(* CoDeSys 2.3.9.35 project: PACMAN.pro *)
(* Libraries: Util_no_Real.lib 1.6.07 09:41:00, Standard.LIB 4.10.05 11:14:46 *)

(* Global variable list: Global_Variables *)
VAR_GLOBAL
    hoz: INT;
    ver: INT;
	MAPA: ARRAY[0..20, 0..15] OF BOOL;
	Mapa_Punkty: ARRAY[0..20, 0..15] OF BOOL;
	Wolne_Prawo: BOOL;
	Wolne_Lewo: BOOL;
	Wolne_Dol: BOOL;
	Wolne_Gora: BOOL;
	Otwarte: BOOL := TRUE;
	Kierunek: INT := 1;
 B_Prawo : BOOL := TRUE;
   B_Lewo  : BOOL;
   B_Dol   : BOOL;
   B_Gora  : BOOL;

END_VAR

(* POU PLC_PRG, LD *)
PROGRAM PLC_PRG
VAR
	S1: BOOL;
	S3: BOOL;
	res: BOOL;
	S2: BOOL;
	S4: BOOL;
	C3: CTUD;
	W1: BOOL;
	C4: CTUD;
	Ruch_Lewo: BOOL;
	Ruch_Dol: BOOL;
	DUMMY: BOOL;
	M1:MAPA;
	Ruch_Gora: BOOL;
	T_Ani: TON;
	C_Ani: CTU;
	SR1: SR;
	Reset_SR1: BOOL;
	SR2: SR;
	Reset_SR2: BOOL;
	SR3: SR;
	Reset_SR3: BOOL;
	Reset_SR4: BOOL;
	SR4: SR;
	T_Ruch: TON;
END_VAR
_LD_ (* Ladder Diagram *)
NETWORK 1
	M1:MAPA()
NETWORK 2
	*
		EN --- ???:OBLICZ_KOLIZJE() => DUMMY
NETWORK 3
	[/T_Ruch.Q] - T_Ruch:TON(IN: *, PT: T#200ms)
NETWORK 4
	[/T_Ruch.Q] - [B_Dol] - [Wolne_Dol] - C3:CTUD(CU: *, CD: Ruch_Gora, RESET: res, LOAD: FALSE, PV: 20, CV => ver)
NETWORK 5
	[/T_Ruch.Q] - [B_Gora] - [Wolne_Gora] --- (Ruch_Gora)
NETWORK 6
	[/T_Ruch.Q] - [B_Prawo] - [Wolne_Prawo] - C4:CTUD(CU: *, CD: Ruch_Lewo, RESET: res, LOAD: FALSE, PV: 15, CV => hoz)
NETWORK 7
	[/T_Ruch.Q] - [B_Lewo] - [Wolne_Lewo] --- (Ruch_Lewo)
NETWORK 8
	[/T_Ani.Q] - T_Ani:TON(IN: *, PT: T#20ms)
NETWORK 9
	[T_Ani.Q] - C_Ani:CTU(CU: *, RESET: C_Ani.Q, PV: 2)
NETWORK 10
	[/C_Ani.CV.0] --- (Otwarte)
NETWORK 11
	[S1] - SR1:SR(SET1: *, RESET: Reset_SR1) --- (B_Prawo)
NETWORK 12
	{ [S2] | [S3] | [S4] } --- (Reset_SR1)
NETWORK 13
	[S2] - SR2:SR(SET1: *, RESET: Reset_SR2) --- (B_Lewo)
NETWORK 14
	{ [S1] | [S3] | [S4] } --- (Reset_SR2)
NETWORK 15
	[S3] - SR3:SR(SET1: *, RESET: Reset_SR3) --- (B_Dol)
NETWORK 16
	{ [S1] | [S2] | [S4] } --- (Reset_SR3)
NETWORK 17
	[S4] - SR4:SR(SET1: *, RESET: Reset_SR4) --- (B_Gora)
NETWORK 18
	{ [S1] | [S2] | [S3] } --- (Reset_SR4)
NETWORK 19
	[Mapa_Punkty[hoz, ver]] --- (R Mapa_Punkty[hoz, ver])
_END_LD_
(* the same logic as Structured Text *)
(* Network 1 *)
M1();
(* Network 2: see the listing above *)
(* Network 3 *)
T_Ruch(IN := NOT T_Ruch.Q, PT := T#200ms);
(* Network 4 *)
C3(CU := NOT T_Ruch.Q AND B_Dol AND Wolne_Dol, CD := Ruch_Gora, RESET := res, LOAD := FALSE, PV := 20);
ver := C3.CV;
(* Network 5 *)
Ruch_Gora := NOT T_Ruch.Q AND B_Gora AND Wolne_Gora;
(* Network 6 *)
C4(CU := NOT T_Ruch.Q AND B_Prawo AND Wolne_Prawo, CD := Ruch_Lewo, RESET := res, LOAD := FALSE, PV := 15);
hoz := C4.CV;
(* Network 7 *)
Ruch_Lewo := NOT T_Ruch.Q AND B_Lewo AND Wolne_Lewo;
(* Network 8 *)
T_Ani(IN := NOT T_Ani.Q, PT := T#20ms);
(* Network 9 *)
C_Ani(CU := T_Ani.Q, RESET := C_Ani.Q, PV := 2);
(* Network 10 *)
Otwarte := NOT C_Ani.CV.0;
(* Network 11 *)
SR1(SET1 := S1, RESET := Reset_SR1);
B_Prawo := SR1.Q1;
(* Network 12 *)
Reset_SR1 := S2 OR S3 OR S4;
(* Network 13 *)
SR2(SET1 := S2, RESET := Reset_SR2);
B_Lewo := SR2.Q1;
(* Network 14 *)
Reset_SR2 := S1 OR S3 OR S4;
(* Network 15 *)
SR3(SET1 := S3, RESET := Reset_SR3);
B_Dol := SR3.Q1;
(* Network 16 *)
Reset_SR3 := S1 OR S2 OR S4;
(* Network 17 *)
SR4(SET1 := S4, RESET := Reset_SR4);
B_Gora := SR4.Q1;
(* Network 18 *)
Reset_SR4 := S1 OR S2 OR S3;
(* Network 19 *)
IF Mapa_Punkty[hoz, ver] THEN Mapa_Punkty[hoz, ver] := FALSE; END_IF;
END_PROGRAM

(* POU MAPA, ST *)
FUNCTION_BLOCK MAPA
VAR
    i: INT;
    j: INT;
    Init_Done: BOOL := FALSE;

END_VAR
IF NOT Init_Done THEN

    (* ======================= *)
    (* 1. RYSOWANIE ŒCIAN      *)
    (* ======================= *)

    FOR i := 0 TO 20 DO
        Mapa[i, 0] := TRUE;
        Mapa[i, 15] := TRUE;
    END_FOR
    
    FOR j := 0 TO 15 DO
        Mapa[0, j] := TRUE;
        MAPA[20, j] := TRUE;
    END_FOR

    Mapa[0, 0] := FALSE;
    Mapa[1, 0] := FALSE;
    Mapa[0, 1] := FALSE;
    Mapa[2, 0] := FALSE;
    Mapa[0, 2] := FALSE;
    Mapa[3, 0] := FALSE;
    Mapa[0, 3] := FALSE;
    Mapa[0, 4] := FALSE;
    Mapa[0, 5] := FALSE;
    Mapa[0, 6] := FALSE;
    Mapa[0, 7] := FALSE;
    Mapa[0, 8] := FALSE;

    Mapa[1, 4] := FALSE;
    Mapa[2, 4] := FALSE;
    Mapa[2, 3] := FALSE;
    Mapa[2, 2] := FALSE;
    Mapa[3, 2] := FALSE;
    
    Mapa[1, 3] := TRUE;
    Mapa[1, 2] := TRUE;
    Mapa[1, 1] := TRUE;
    Mapa[2, 1] := TRUE;

    Mapa[1, 5] := TRUE;
    Mapa[1, 6] := TRUE;
    Mapa[1, 7] := TRUE;
    Mapa[2, 7] := TRUE;
    Mapa[3, 5] := TRUE;
    Mapa[4, 5] := TRUE;
    Mapa[3, 3] := TRUE;
    Mapa[4, 3] := TRUE;
    Mapa[4, 7] := TRUE;
    Mapa[4, 8] := TRUE;

    Mapa[6, 1] := TRUE;
    Mapa[7, 1] := TRUE;
    Mapa[8, 1] := TRUE;
    Mapa[9, 1] := TRUE;
    Mapa[10, 1] := TRUE;
    Mapa[11, 1] := TRUE;
    Mapa[12, 1] := TRUE;

    Mapa[6, 3] := TRUE;
    Mapa[7, 3] := TRUE;
    Mapa[11, 3] := TRUE;
    Mapa[12, 3] := TRUE;
    Mapa[6, 4] := TRUE;
    Mapa[12, 4] := TRUE;

    Mapa[6, 5] := TRUE;
    Mapa[7, 5] := TRUE;
    Mapa[8, 5] := TRUE;
    Mapa[9, 5] := TRUE;
    Mapa[10, 5] := TRUE;
    Mapa[11, 5] := TRUE;
    Mapa[12, 5] := TRUE;

    Mapa[6, 7] := TRUE;
    Mapa[7, 7] := TRUE;
    Mapa[8, 7] := TRUE;
    Mapa[9, 7] := TRUE;
    Mapa[10, 7] := TRUE;
    Mapa[11, 7] := TRUE;
    Mapa[12, 7] := TRUE;

    Mapa[14, 0] := TRUE;
    Mapa[14, 1] := TRUE;
    Mapa[14, 3] := TRUE;
    Mapa[14, 5] := TRUE;
    Mapa[15, 5] := TRUE;
    Mapa[14, 7] := TRUE;
    Mapa[14, 8] := TRUE;
    Mapa[15, 3] := TRUE;
    Mapa[16, 1] := TRUE;
    Mapa[16, 7] := TRUE;

    Mapa[17, 1] := TRUE;
    Mapa[17, 2] := TRUE;
    Mapa[17, 3] := TRUE;
    Mapa[17, 5] := TRUE;
    Mapa[17, 6] := TRUE;
    Mapa[17, 7] := TRUE;
    
    Mapa[4, 1] := TRUE;

    Mapa[5, 0] := FALSE;
    Mapa[6, 0] := FALSE;
    Mapa[7, 0] := FALSE;
    Mapa[8, 0] := FALSE;
    Mapa[9, 0] := FALSE;
    Mapa[10, 0] := FALSE;
    Mapa[11, 0] := FALSE;
    Mapa[12, 0] := FALSE;
    Mapa[13, 0] := FALSE;
    Mapa[15, 0] := FALSE;
    Mapa[16, 0] := FALSE;
    Mapa[17, 0] := FALSE;
    Mapa[18, 0] := FALSE;


    Mapa[1, 9] := TRUE;
    Mapa[2, 9] := TRUE;
    Mapa[3, 9] := TRUE;
    Mapa[4, 9] := TRUE;
    Mapa[5, 9] := TRUE;
    Mapa[6, 9] := TRUE;
    Mapa[7, 9] := TRUE;
    Mapa[8, 9] := TRUE;
    Mapa[9, 9] := TRUE;
    Mapa[10, 9] := TRUE;
    Mapa[11, 9] := TRUE;
    Mapa[12, 9] := TRUE;
    Mapa[13, 9] := TRUE;
    Mapa[14, 9] := TRUE;
    Mapa[15, 9] := TRUE;
    Mapa[16, 9] := TRUE;
    Mapa[17, 9] := TRUE;
    Mapa[18, 9] := TRUE;
    Mapa[19, 9] := TRUE;

    Mapa[19, 1] := TRUE;
    Mapa[19, 2] := TRUE;
    Mapa[19, 3] := TRUE;
    Mapa[19, 4] := TRUE;
    Mapa[19, 5] := TRUE;
    Mapa[19, 6] := TRUE;
    Mapa[19, 7] := TRUE;
    Mapa[19, 8] := TRUE;

    (* ======================= *)
    (* 2. RYSOWANIE PUNKTÓW    *)
    (* ======================= *)
    
	Mapa_Punkty[0, 2] := TRUE;
	Mapa_Punkty[0, 3] := TRUE;
	Mapa_Punkty[0, 4] := TRUE;
	Mapa_Punkty[0, 5] := TRUE;
	Mapa_Punkty[0, 6] := TRUE;
	Mapa_Punkty[0, 7] := TRUE;
	Mapa_Punkty[0, 8] := TRUE;
	Mapa_Punkty[1, 8] := TRUE;
	Mapa_Punkty[2, 8] := TRUE;
	Mapa_Punkty[3, 8] := TRUE;
	Mapa_Punkty[3, 7] := TRUE;
	Mapa_Punkty[3, 6] := TRUE;
	Mapa_Punkty[4, 6] := TRUE;
	Mapa_Punkty[5, 6] := TRUE;
	Mapa_Punkty[6, 6] := TRUE;
	Mapa_Punkty[7, 6] := TRUE;
	Mapa_Punkty[8, 6] := TRUE;
	Mapa_Punkty[9, 6] := TRUE;
	Mapa_Punkty[10, 6] := TRUE;
	Mapa_Punkty[11,6] := TRUE;
	Mapa_Punkty[12, 6] := TRUE;
	Mapa_Punkty[13, 6] := TRUE;
	Mapa_Punkty[14, 6] := TRUE;
	Mapa_Punkty[15, 6] := TRUE;
	Mapa_Punkty[16, 6] := TRUE;
	
	Mapa_Punkty[6, 8] := TRUE;
	Mapa_Punkty[7, 8] := TRUE;
	Mapa_Punkty[8, 8] := TRUE;
	Mapa_Punkty[9, 8] := TRUE;
	Mapa_Punkty[10, 8] := TRUE;
	Mapa_Punkty[11, 8] := TRUE;
	Mapa_Punkty[12, 8] := TRUE;
	Mapa_Punkty[13, 8] := TRUE;
	Mapa_Punkty[5, 8] := TRUE;
	
	Mapa_Punkty[6, 0] := TRUE;
	Mapa_Punkty[7, 0] := TRUE;
	Mapa_Punkty[8, 0] := TRUE;
	Mapa_Punkty[9, 0] := TRUE;
	Mapa_Punkty[10, 0] := TRUE;
	Mapa_Punkty[11, 0] := TRUE;
	Mapa_Punkty[12, 0] := TRUE;
	Mapa_Punkty[13, 0] := TRUE;
	Mapa_Punkty[5, 0] := TRUE;
	
	Mapa_Punkty[18, 0] := TRUE;
	Mapa_Punkty[18, 1] := TRUE;
	Mapa_Punkty[18, 2] := TRUE;
	Mapa_Punkty[18, 3] := TRUE;
	Mapa_Punkty[18, 4] := TRUE;
	Mapa_Punkty[18, 5] := TRUE;
	Mapa_Punkty[18, 6] := TRUE;
	Mapa_Punkty[18, 7] := TRUE;
	Mapa_Punkty[18, 8] := TRUE;
	
	Mapa_Punkty[2, 2] := TRUE;
	Mapa_Punkty[3, 2] := TRUE;
	Mapa_Punkty[4, 2] := TRUE;
	Mapa_Punkty[5, 2] := TRUE;
	Mapa_Punkty[6, 2] := TRUE;
	Mapa_Punkty[7, 2] := TRUE;
	Mapa_Punkty[8, 2] := TRUE;
	Mapa_Punkty[9, 2] := TRUE;
	Mapa_Punkty[10, 2] := TRUE;
	Mapa_Punkty[11, 2] := TRUE;
	Mapa_Punkty[12, 2] := TRUE;
	Mapa_Punkty[13, 2] := TRUE;
	Mapa_Punkty[14, 2] := TRUE;
	Mapa_Punkty[15, 2] := TRUE;
	Mapa_Punkty[16, 2] := TRUE;
	
	Mapa_Punkty[2, 3] := TRUE;
	Mapa_Punkty[2, 4] := TRUE;
	Mapa_Punkty[2, 5] := TRUE;
	Mapa_Punkty[2, 6] := TRUE;
	
	Mapa_Punkty[5, 0] := TRUE;
	Mapa_Punkty[5, 1] := TRUE;
	Mapa_Punkty[5, 3] := TRUE;
	Mapa_Punkty[5, 4] := TRUE;
	Mapa_Punkty[5, 5] := TRUE;
	Mapa_Punkty[5, 7] := TRUE;
	Mapa_Punkty[5, 8] := TRUE;
	Mapa_Punkty[3, 4] := TRUE;
	Mapa_Punkty[4, 4] := TRUE;
	
	Mapa_Punkty[8, 3] := TRUE;
	Mapa_Punkty[9, 3] := TRUE;
	Mapa_Punkty[10, 3] := TRUE;
	
	Mapa_Punkty[7,4] := TRUE;
	Mapa_Punkty[8,4] := TRUE;
	Mapa_Punkty[9,4] := TRUE;
	Mapa_Punkty[10,4] := TRUE;
	Mapa_Punkty[11,4] := TRUE;
	
	Mapa_Punkty[13,1] := TRUE;
	Mapa_Punkty[13,3] := TRUE;
	Mapa_Punkty[13,4] := TRUE;
	Mapa_Punkty[13,5] := TRUE;
	Mapa_Punkty[13,7] := TRUE;
	
	Mapa_Punkty[13,4] := TRUE;
	Mapa_Punkty[14,4] := TRUE;
	Mapa_Punkty[15,4] := TRUE;
	Mapa_Punkty[16,4] := TRUE;
	Mapa_Punkty[17,4] := TRUE;
	
	Mapa_Punkty[16,3] := TRUE;
	Mapa_Punkty[16,5] := TRUE;
	
	Mapa_Punkty[15,0] := TRUE;
	Mapa_Punkty[16,0] := TRUE;
	Mapa_Punkty[17,0] := TRUE;
	Mapa_Punkty[15,8] := TRUE;
	Mapa_Punkty[16,8] := TRUE;
	Mapa_Punkty[17,8] := TRUE;
	Mapa_Punkty[15,1] := TRUE;
	Mapa_Punkty[1,4] := TRUE;
	Mapa_Punkty[15,7] := TRUE;
	
	Mapa_Punkty[1,0] := TRUE;
	Mapa_Punkty[2,0] := TRUE;
	Mapa_Punkty[3,0] := TRUE;
	Mapa_Punkty[3,1] := TRUE;

    Init_Done := TRUE;

END_IF
END_FUNCTION_BLOCK

(* POU OBLICZ_KOLIZJE, ST *)
PROGRAM OBLICZ_KOLIZJE
VAR
END_VAR
Wolne_Prawo := FALSE;
Wolne_Lewo := FALSE;
Wolne_Gora := FALSE;
Wolne_Dol := FALSE;

IF hoz < 20 THEN
    IF Mapa[hoz + 1, ver] = FALSE THEN
        Wolne_Prawo := TRUE;
    END_IF
END_IF


IF hoz > 0 THEN
    IF Mapa[hoz - 1, ver] = FALSE THEN
        Wolne_Lewo := TRUE;
    END_IF
END_IF

IF ver < 15 THEN
    IF Mapa[hoz, ver + 1] = FALSE THEN
        Wolne_Dol := TRUE;
    END_IF
END_IF

IF ver > 0 THEN
    IF Mapa[hoz, ver - 1] = FALSE THEN
        Wolne_Gora := TRUE;
    END_IF
END_IF
END_PROGRAM

(* Visualisation GRA
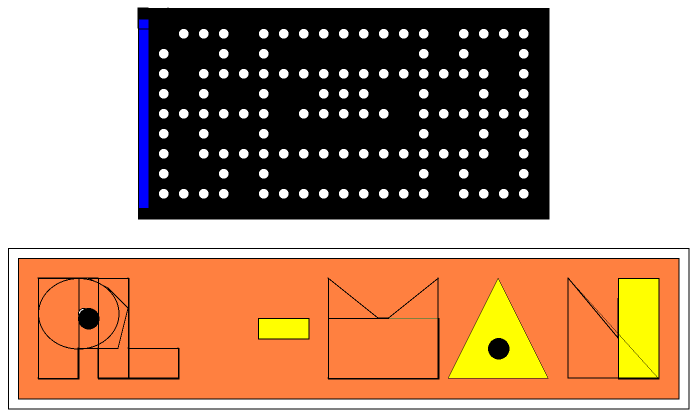
ellipse at (180,150)-(191,161): invisible if NOT Mapa_Punkty[0, 1]
ellipse at (180,190)-(191,201): invisible if NOT Mapa_Punkty[0, 3]
ellipse at (180,210)-(191,221): invisible if NOT Mapa_Punkty[0, 4]
ellipse at (180,230)-(191,241): invisible if NOT Mapa_Punkty[0,5]
ellipse at (180,250)-(191,261): invisible if NOT Mapa_Punkty[0,6]
ellipse at (180,270)-(191,281): invisible if NOT Mapa_Punkty[0,7]
ellipse at (180,290)-(191,301): invisible if NOT Mapa_Punkty[0,8]
ellipse at (200,290)-(211,301): invisible if NOT Mapa_Punkty[1,8]
ellipse at (220,290)-(231,301): invisible if NOT Mapa_Punkty[2,8]
ellipse at (240,290)-(251,301): invisible if NOT Mapa_Punkty[3,8]
ellipse at (240,270)-(251,281): invisible if NOT Mapa_Punkty[3,7]
ellipse at (240,250)-(251,261): invisible if NOT Mapa_Punkty[3,6]
ellipse at (220,250)-(231,261): invisible if NOT Mapa_Punkty[2,6]
ellipse at (260,250)-(271,261): invisible if NOT Mapa_Punkty[4,6]
ellipse at (280,250)-(291,261): invisible if NOT Mapa_Punkty[5,6]
ellipse at (300,250)-(311,261): invisible if NOT Mapa_Punkty[6,6]
ellipse at (320,250)-(331,261): invisible if NOT Mapa_Punkty[7,6]
ellipse at (340,250)-(351,261): invisible if NOT Mapa_Punkty[8,6]
ellipse at (360,250)-(371,261): invisible if NOT Mapa_Punkty[9,6]
ellipse at (380,250)-(391,261): invisible if NOT Mapa_Punkty[10,6]
ellipse at (400,250)-(411,261): invisible if NOT Mapa_Punkty[11,6]
ellipse at (420,250)-(431,261): invisible if NOT Mapa_Punkty[12,6]
ellipse at (440,250)-(451,261): invisible if NOT Mapa_Punkty[13,6]
ellipse at (460,250)-(471,261): invisible if NOT Mapa_Punkty[14,6]
ellipse at (480,250)-(491,261): invisible if NOT Mapa_Punkty[15,6]
ellipse at (500,250)-(511,261): invisible if NOT Mapa_Punkty[16,6]
ellipse at (280,290)-(291,301): invisible if NOT Mapa_Punkty[5,8]
ellipse at (300,290)-(311,301): invisible if NOT Mapa_Punkty[6,8]
ellipse at (320,290)-(331,301): invisible if NOT Mapa_Punkty[7,8]
ellipse at (340,290)-(351,301): invisible if NOT Mapa_Punkty[8,8]
ellipse at (360,290)-(371,301): invisible if NOT Mapa_Punkty[9,8]
ellipse at (380,290)-(391,301): invisible if NOT Mapa_Punkty[10,8]
ellipse at (400,290)-(411,301): invisible if NOT Mapa_Punkty[11,8]
ellipse at (420,290)-(431,301): invisible if NOT Mapa_Punkty[12,8]
ellipse at (440,290)-(451,301): invisible if NOT Mapa_Punkty[13,8]
ellipse at (280,130)-(291,141): invisible if NOT Mapa_Punkty[5,0]
ellipse at (300,130)-(311,141): invisible if NOT Mapa_Punkty[6,0]
ellipse at (320,130)-(331,141): invisible if NOT Mapa_Punkty[7,0]
ellipse at (340,130)-(351,141): invisible if NOT Mapa_Punkty[8,0]
ellipse at (360,130)-(371,141): invisible if NOT Mapa_Punkty[9,0]
ellipse at (380,130)-(391,141): invisible if NOT Mapa_Punkty[10,0]
ellipse at (400,130)-(411,141): invisible if NOT Mapa_Punkty[11,0]
ellipse at (420,130)-(431,141): invisible if NOT Mapa_Punkty[12,0]
ellipse at (440,130)-(451,141): invisible if NOT Mapa_Punkty[13,0]
ellipse at (540,150)-(551,161): invisible if NOT Mapa_Punkty[18,1]
ellipse at (540,170)-(551,181): invisible if NOT Mapa_Punkty[18,2]
ellipse at (540,190)-(551,201): invisible if NOT Mapa_Punkty[18,3]
ellipse at (540,210)-(551,221): invisible if NOT Mapa_Punkty[18,4]
ellipse at (540,230)-(551,241): invisible if NOT Mapa_Punkty[18,5]
ellipse at (540,250)-(551,261): invisible if NOT Mapa_Punkty[18,6]
ellipse at (540,270)-(551,281): invisible if NOT Mapa_Punkty[18,7]
ellipse at (540,290)-(551,301): invisible if NOT Mapa_Punkty[18,8]
ellipse at (540,130)-(551,141): invisible if NOT Mapa_Punkty[18, 0]
ellipse at (220,170)-(231,181): invisible if NOT Mapa_Punkty[2,2]
ellipse at (240,170)-(251,181): invisible if NOT Mapa_Punkty[3,2]
ellipse at (260,170)-(271,181): invisible if NOT Mapa_Punkty[4,2]
ellipse at (280,170)-(291,181): invisible if NOT Mapa_Punkty[5,2]
ellipse at (300,170)-(311,181): invisible if NOT Mapa_Punkty[6,2]
ellipse at (320,170)-(331,181): invisible if NOT Mapa_Punkty[7,2]
ellipse at (340,170)-(351,181): invisible if NOT Mapa_Punkty[8,2]
ellipse at (360,170)-(371,181): invisible if NOT Mapa_Punkty[9,2]
ellipse at (380,170)-(391,181): invisible if NOT Mapa_Punkty[10,2]
ellipse at (400,170)-(411,181): invisible if NOT Mapa_Punkty[11,2]
ellipse at (420,170)-(431,181): invisible if NOT Mapa_Punkty[12,2]
ellipse at (440,170)-(451,181): invisible if NOT Mapa_Punkty[13,2]
ellipse at (460,170)-(471,181): invisible if NOT Mapa_Punkty[14,2]
ellipse at (480,170)-(491,181): invisible if NOT Mapa_Punkty[15,2]
ellipse at (500,170)-(511,181): invisible if NOT Mapa_Punkty[16,2]
ellipse at (220,190)-(231,201): invisible if NOT Mapa_Punkty[2,3]
ellipse at (220,210)-(231,221): invisible if NOT Mapa_Punkty[2,4]
ellipse at (220,230)-(231,241): invisible if NOT Mapa_Punkty[2,5]
ellipse at (280,150)-(291,161): invisible if NOT Mapa_Punkty[5,1]
ellipse at (280,190)-(291,201): invisible if NOT Mapa_Punkty[5,3]
ellipse at (280,210)-(291,221): invisible if NOT Mapa_Punkty[5,4]
ellipse at (280,230)-(291,241): invisible if NOT Mapa_Punkty[5,5]
ellipse at (280,270)-(291,281): invisible if NOT Mapa_Punkty[5,7]
ellipse at (240,210)-(251,221): invisible if NOT Mapa_Punkty[3,4]
ellipse at (260,210)-(271,221): invisible if NOT Mapa_Punkty[4,4]
ellipse at (320,210)-(331,221): invisible if NOT Mapa_Punkty[7,4]
ellipse at (340,210)-(351,221): invisible if NOT Mapa_Punkty[8,4]
ellipse at (360,210)-(371,221): invisible if NOT Mapa_Punkty[9,4]
ellipse at (380,210)-(391,221): invisible if NOT Mapa_Punkty[10,4]
ellipse at (400,210)-(411,221): invisible if NOT Mapa_Punkty[11,4]
ellipse at (340,190)-(351,201): invisible if NOT Mapa_Punkty[8,3]
ellipse at (360,190)-(371,201): invisible if NOT Mapa_Punkty[9,3]
ellipse at (380,190)-(391,201): invisible if NOT Mapa_Punkty[10,3]
ellipse at (440,150)-(451,161): invisible if NOT Mapa_Punkty[13,1]
ellipse at (440,190)-(451,201): invisible if NOT Mapa_Punkty[13,3]
ellipse at (440,210)-(451,221): invisible if NOT Mapa_Punkty[13,4]
ellipse at (440,230)-(451,241): invisible if NOT Mapa_Punkty[13,5]
ellipse at (440,270)-(451,281): invisible if NOT Mapa_Punkty[13,7]
ellipse at (460,210)-(471,221): invisible if NOT Mapa_Punkty[14,4]
ellipse at (480,210)-(491,221): invisible if NOT Mapa_Punkty[15,4]
ellipse at (500,210)-(511,221): invisible if NOT Mapa_Punkty[16,4]
ellipse at (520,210)-(531,221): invisible if NOT Mapa_Punkty[17,4]
ellipse at (500,230)-(511,241): invisible if NOT Mapa_Punkty[16,5]
ellipse at (500,190)-(511,201): invisible if NOT Mapa_Punkty[16,3]
ellipse at (480,130)-(491,141): invisible if NOT Mapa_Punkty[15, 0]
ellipse at (500,130)-(511,141): invisible if NOT Mapa_Punkty[16, 0]
ellipse at (520,130)-(531,141): invisible if NOT Mapa_Punkty[17, 0]
ellipse at (480,290)-(491,301): invisible if NOT Mapa_Punkty[15,8]
ellipse at (500,290)-(511,301): invisible if NOT Mapa_Punkty[16,8]
ellipse at (520,290)-(531,301): invisible if NOT Mapa_Punkty[17,8]
ellipse at (480,150)-(491,161): invisible if NOT Mapa_Punkty[15,1]
ellipse at (480,270)-(491,281): invisible if NOT Mapa_Punkty[15,7]
ellipse at (200,210)-(211,221): invisible if NOT Mapa_Punkty[1,4]
ellipse at (180,170)-(191,181): invisible if NOT Mapa_Punkty[0,2]
ellipse at (200,130)-(211,141): invisible if NOT Mapa_Punkty[1,0]
ellipse at (220,130)-(231,141): invisible if NOT Mapa_Punkty[2,0]
ellipse at (240,130)-(251,141): invisible if NOT Mapa_Punkty[3,0]
ellipse at (240,150)-(251,161): invisible if NOT Mapa_Punkty[3,1]
56 more shapes without text or variables
6 elements of other kinds (tables, trends, ...) not read
*)
